FUNCTION_BLOCK FB_GCWaferReceiveService EXTENDS FB_ServiceBase
VAR_INPUT
	Param : ST_WaferTransferParam;
	SpinAxis_BaseUnit : I_Axis_BaseUnit;
	LiftPinAxis_BaseUnit : I_Axis_BaseUnit;
END_VAR

VAR_IN_OUT
	// Shared with the opposite direction; arbitration belongs to the future transfer flow.
	MaterialInfo : ST_MaterialInfo;
END_VAR

VAR_OUTPUT
	SignalOut : ST_TransferHandshakeSignal;
END_VAR

M_UpdateService(CompletionBehavior := E_ServiceCompletionBehavior.NaturalCompletion);

METHOD PROTECTED H_OnAborting : E_PackMLHookResult
VAR_INPUT
	bFirstScan : BOOL;
END_VAR
// TODO: Implement abort cleanup and material reconciliation for an interrupted transfer.
// The skeleton acquires no resources and issues no hardware commands.
H_OnAborting := E_PackMLHookResult.Done;
END_METHOD

METHOD PROTECTED H_OnCompleting : E_PackMLHookResult
VAR_INPUT
	bFirstScan : BOOL;
END_VAR
// TODO: Finish handshake cleanup and release resources after confirmed completion.
H_OnCompleting := E_PackMLHookResult.Done;
END_METHOD

METHOD PROTECTED H_OnExecute : E_PackMLHookResult
VAR_INPUT
	bFirstScan : BOOL;
END_VAR
// TODO: Implement receiving into GC, handshake sequencing, and timeout handling.
// TransferReady advertises Endpoint availability; SignalOut.Ready is a handshake signal.
// TODO: Update MaterialInfo with the received MaterialContext only after confirmed receive completion.
// Keep the skeleton active until Stop/Abort; do not report a completed transfer.
H_OnExecute := E_PackMLHookResult.Busy;
END_METHOD

METHOD PROTECTED H_OnResetting : E_PackMLHookResult
VAR_INPUT
	bFirstScan : BOOL;
END_VAR
MEMSET(ADR(Status.ErrorList), 0, SIZEOF(Status.ErrorList));
// TODO: Reset transfer-local state without unconditionally clearing the Station material.
H_OnResetting := E_PackMLHookResult.Done;
END_METHOD

METHOD PROTECTED H_OnStarting : E_PackMLHookResult
VAR_INPUT
	bFirstScan : BOOL;
END_VAR
// TODO: Validate Param against StationId, latch transfer data, and reserve resources.
H_OnStarting := E_PackMLHookResult.Done;
END_METHOD

METHOD PROTECTED H_OnStopping : E_PackMLHookResult
VAR_INPUT
	bFirstScan : BOOL;
END_VAR
// TODO: Withdraw handshake/motion requests and complete owned-resource cleanup.
// The skeleton acquires no resources and issues no hardware commands.
H_OnStopping := E_PackMLHookResult.Done;
END_METHOD

END_FUNCTION_BLOCK

(* stored: Version 1.1.0.1, ProductVersion 3.1.4026.18
   POU FB_GCWaferReceiveService: Id {31c0f8a3-2bb7-4853-987f-7b1795d30426}, SpecialFunc None
   Folder StateAction: Id {60d1dd31-2224-4849-ae56-5d896fbf2a68}
   Method H_OnAborting: Id {f6237217-291f-47f3-85aa-1d639fca1749}
   Method H_OnCompleting: Id {45ff17a5-ca23-45cb-ab02-4b17bc7ba00f}
   Method H_OnExecute: Id {03bc22fb-3dc2-4986-a5e4-87270d37378e}
   Method H_OnResetting: Id {2d387bfa-b920-4024-aa27-c9ea79ce1983}
   Method H_OnStarting: Id {b779e2ff-ae11-4e0a-a9e3-c1b8c4be40d0}
   Method H_OnStopping: Id {434a4009-61a5-420a-a161-ff8cb745394e} *)
